// Mitsubishi GX Developer project: 模拟抢答器   PLC: FX3U

PROGRAM MAIN
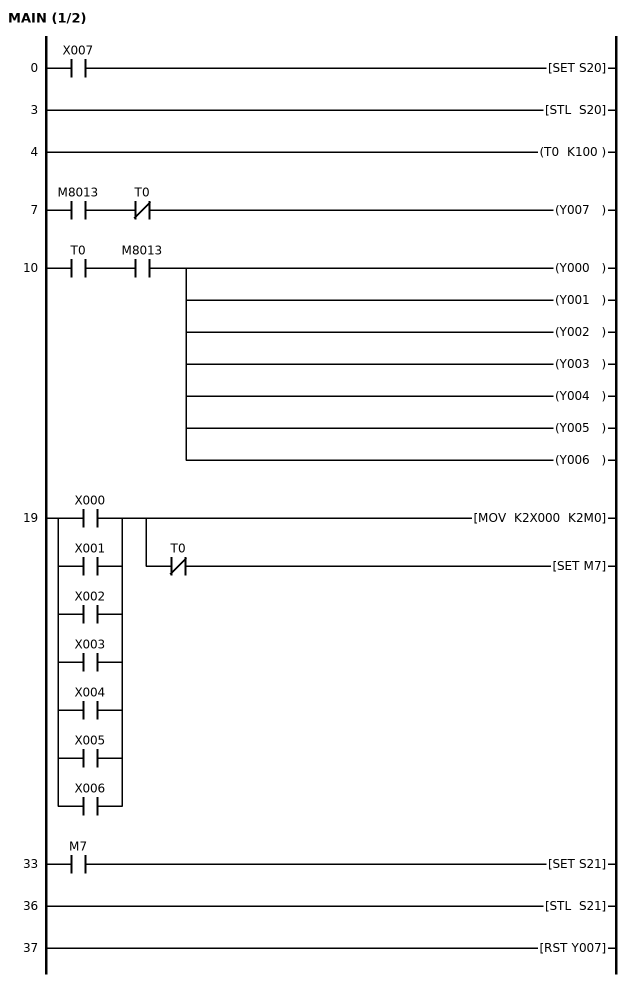
0     LD      X007
      SET     S20
3     STL     S20
4     OUT     T0 K100
7     LD      M8013
      ANI     T0
      OUT     Y007
10    LD      T0
      AND     M8013
      OUT     Y000
      OUT     Y001
      OUT     Y002
      OUT     Y003
      OUT     Y004
      OUT     Y005
      OUT     Y006
19    LD      X000
      OR      X001
      OR      X002
      OR      X003
      OR      X004
      OR      X005
      OR      X006
      MOV     K2X000 K2M0
      ANI     T0
      SET     M7
33    LD      M7
      SET     S21
36    STL     S21
37    RST     Y007
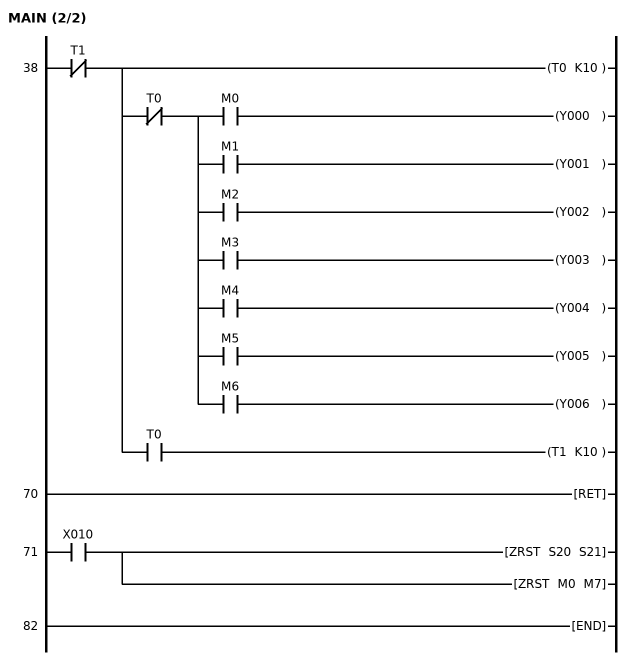
38    LDI     T1
      OUT     T0 K10
      MPS
      ANI     T0
      MPS
      AND     M0
      OUT     Y000
      MRD
      AND     M1
      OUT     Y001
      MRD
      AND     M2
      OUT     Y002
      MRD
      AND     M3
      OUT     Y003
      MRD
      AND     M4
      OUT     Y004
      MRD
      AND     M5
      OUT     Y005
      MPP
      AND     M6
      OUT     Y006
      MPP
      AND     T0
      OUT     T1 K10
70    RET
71    LD      X010
      ZRST    S20 S21
      ZRST    M0 M7
82    END
END_PROGRAM
